Fanuc KAREL source: kt00369.KL

-- PROVISIONAL review KL for V1013-1; original PC SHA256 1aab6ac64b91335ff9e2b58386e289a7d15b806000a49ac7ab307cda12c6bd85
-- Incomplete behavior may be omitted. Consult companion uncertainty JSON. Do not deploy.
PROGRAM KT00369
%NOLOCKGROUP
VAR
  R1 : REAL
  I2 : INTEGER
  OUT : BOOLEAN
BEGIN
  -- UNRESOLVED_PC offsets 5-16; opcodes 2E,23
  -- UNRESOLVED_PC offsets 21-32; opcodes 2E,23
  -- UNRESOLVED_PC offsets 37-57; opcodes 21,21,64,70,23
  -- UNRESOLVED_PC offsets 62-66; opcodes 7F
END KT00369
